# B&R Automation Studio project Lab3
Automation Studio 4.5.2.102

## Configuration SampleText

### IoMap.iom - 4PP065_0571_P74/IoMap.iom
```iecst
VAR_CONFIG
	::SDCAxisCtr:pwm_period AT %QW."X20MM4456".PeriodDurationPWM;
	::SDCAxisCtr:axis_X.pwm_value AT %QW."X20MM4456".PulseWidthCurrentPWM01;
	::SDCAxisCtr:axis_X.reset_error AT %QX."X20MM4456".ClearError01;
	::SDCAxisCtr:axis_X.reset_counter AT %QX."X20MM4456".ResetCounter01;
	::SDCAxisCtr:axis_X.counter AT %IW."X20MM4456".Counter01;
	::SDCAxisCtr:axis_X.endswitch_b_reached AT %IX."X20MM4456".StatusInput03;
	::SDCAxisCtr:axis_X.endswitch_a_reached AT %IX."X20MM4456".StatusInput04;
	::SDCAxisCtr:coil_pwm_value AT %QW."X20MM4456".PulseWidthCurrentPWM04;
	::SDCAxisCtr:axis_X.direction AT %IX."X20DI9371".DigitalInput01;
	::SDCAxisCtr:axis_X.button_b AT %IX."X20DI9371".DigitalInput02;
	::SDCAxisCtr:axis_X.button_a AT %IX."X20DI9371".DigitalInput03;
	::SDCAxisCtr:coil_powered AT %IX."X20DI9371".DigitalInput04;
	::SDCAxisCt1:axis_Y.pwm_value AT %QW."X20MM4456".PulseWidthCurrentPWM02;
	::SDCAxisCt1:axis_Y.reset_error AT %QX."X20MM4456".ClearError02;
	::SDCAxisCt1:axis_Y.reset_counter AT %QX."X20MM4456".ResetCounter02;
	::SDCAxisCt1:axis_Y.counter AT %IW."X20MM4456".Counter02;
	::SDCAxisCt1:axis_Y.endswitch_a_reached AT %IX."X20MM4456".StatusInput07;
	::SDCAxisCt1:axis_Y.endswitch_b_reached AT %IX."X20MM4456".StatusInput08;
	::SDCAxisCt2:axis_Z.pwm_value AT %QW."X20MM4456".PulseWidthCurrentPWM03;
	::SDCAxisCt2:axis_Z.reset_error AT %QX."X20MM4456".ClearError03;
	::SDCAxisCt2:axis_Z.reset_counter AT %QX."X20MM4456".ResetCounter03;
	::SDCAxisCt2:axis_Z.counter AT %IW."X20MM4456".Counter03;
	::SDCAxisCt2:axis_Z.endswitch_a_reached AT %IX."X20MM4456".StatusInput12;
	::SDCAxisCt2:axis_Z.endswitch_b_reached AT %IX."X20MM4456".StatusInput11;
END_VAR
```

### Acp10map1.ncm - 4PP065_0571_P74/Motion/Acp10map1.ncm
```
NcMapping (NcSwId=ACP10, DisabledNodesAreHidden=False)
  NcObject gAxis_X (ModuleAddress=SDC_IF1.ST1, InterfaceType=SDC, Type=ncAXIS, Channel=1, AcoposSimulation=Off, InitParameter=gAxis_X_01, AcoposParameter=gAxis_X_1, AdditionalData=CNC_Enabled="1", Disabled=FALSE, ModuleDisabled=FALSE)
  NcObject gAxis_Y (ModuleAddress=SDC_IF1.ST2, InterfaceType=SDC, Type=ncAXIS, Channel=1, AcoposSimulation=Off, InitParameter=gAxis_YZ_0, AcoposParameter=gAxis_YZ01, AdditionalData=CNC_Enabled="1", Disabled=FALSE)
  NcObject gAxis_Z (ModuleAddress=SDC_IF1.ST3, InterfaceType=SDC, Type=ncAXIS, Channel=1, AcoposSimulation=Off, InitParameter=gAxis_YZ_0, AcoposParameter=gAxis_YZ01, AdditionalData=CNC_Enabled="1", Disabled=FALSE)
```

### Arnc0map.ncm - 4PP065_0571_P74/Motion/Arnc0map.ncm
```
NcMapping (NcSwId=ARNC0)
```

### Arnc0map1.ncm - 4PP065_0571_P74/Motion/Arnc0map1.ncm
```
NcMapping (NcSwId=ARNC0, DisabledNodesAreHidden=False)
  NcObject CNCsys (Type=ncCNCSYS, Channel=1, AcoposSimulation=Off, InitParameter=CncInit, Disabled=FALSE, ModuleDisabled=FALSE)
```

## Logical view

Binary libraries used (declarations not repeated): Runtime, Operator, AsIecCon, astime, sys_lib, asstring, brsystem, AsBrStr, AsIOTime, DataObj, AsArLog, FileIO, AsArProf, AsMem, Arnc0man, Acp10man, Acp10par, NcGlobal, Acp10sim, Acp10sdc, Acp10_MC

### Global.var - Global variables
```iecst
VAR
	gAxis_X : ACP10AXIS_typ := (0);
	gAxis_X_HW : SdcHwCfg_typ := (0);
	gAxis_X_DrvIf : SdcDrvIf16_typ := (0);
	gAxis_X_DiDoIf : SdcDiDoIf_typ := (0);
	gAxis_X_EncIf : SdcEncIf16_typ := (0);
	gAxis_Y : ACP10AXIS_typ := (0);
	gAxis_Y_HW : SdcHwCfg_typ := (0);
	gAxis_Y_DrvIf : SdcDrvIf16_typ := (0);
	gAxis_Y_DiDoIf : SdcDiDoIf_typ := (0);
	gAxis_Y_EncIf : SdcEncIf16_typ := (0);
	gAxis_Z : ACP10AXIS_typ := (0);
	gAxis_Z_HW : SdcHwCfg_typ := (0);
	gAxis_Z_DrvIf : SdcDrvIf16_typ := (0);
	gAxis_Z_DiDoIf : SdcDiDoIf_typ := (0);
	gAxis_Z_EncIf : SdcEncIf16_typ := (0);
	CNCsys : ARNC0CNC_typ := (0);
END_VAR
```

### Package Logical/Libraries - Global libraries

### Library Logical/Libraries/MotrContr (ANSIC)

#### FB_Axis.c
```c
#include <bur/plctypes.h>
#ifdef __cplusplus
	extern "C"
	{
#endif
	#include "MotrContr.h"
#ifdef __cplusplus
	};
#endif
/* TODO: Add your comment here */
void FB_Axis(struct FB_Axis* inst)
{

	/*
	switch(inst->state)
	{
		case unknown:
			if (inst->endswitch_a_reached || inst->button_a)
				inst->state = A;

			if (inst->endswitch_b_reached || inst->button_b)
				inst->state = B;

			if (inst->direction)								//
				inst->state = A_dir;

			if (!inst->direction)								//
				inst->state = B_dir;

			break;

		case B:
			inst->pwm_value = 0;
			inst->reset_error = 1;

			if (!inst->button_b && !inst->endswitch_b_reached)
				inst->state = B_dir;

			if (inst->direction)								//
				inst->state = A_dir;
			break;

		case A:
			inst->pwm_value = 0;
			inst->reset_error = 1;

			if (!inst->button_a && !inst->endswitch_a_reached)
				inst->state = A_dir;

			if (!inst->direction)								//
				inst->state = B_dir;
			break;

		case A_dir:
			inst->pwm_value = inst->u / 24.0 * 32767;			//шим соответственно напряжению с регулятора
			inst->reset_error = 0;
			inst->speed = inst->u / 24.0 * 6500.0;

			if (inst->endswitch_a_reached || inst->button_a)
				inst->state = A;

			if (!inst->direction)								//
				inst->state = B_dir;

			break;

		case B_dir:
			inst->pwm_value = -inst->u / 24.0 * 32767;			//шим соответственно напряжению с регулятора
			inst->reset_error = 0;
			inst->speed = -inst->u / 24.0 * 6500.0;

			if (inst->endswitch_b_reached || inst->button_b)
				inst->state = B;

			if (inst->direction)								//
				inst->state = A_dir;

			break;
	}
	*/

	/*if (inst->endswitch_a_reached || inst->endswitch_b_reached)
	{
		inst->reset_error=1;
	}
	else
	{*/
		inst->pwm_value= inst->u / 24.0 * 32767;//шим соответственно напряжению с регулятора
		//inst->reset_error=0;
	///}
	inst->speed = inst->u / 24.0 * 6500.0;
}
```

### Data object Logical/gAxis_X/gAxis_X_01i (Ax)

#### AxInitAcp10.ax - ACP10 init object for axis
```
InitParameter (Version=5.2.1, NcSwId=ACP10)
  ACP10AXIS_typ:
    dig_in:
      level:
        reference = ncACTIV_HI
        pos_hw_end = ncACTIV_HI
        neg_hw_end = ncACTIV_HI
        trigger1 = ncACTIV_HI
        trigger2 = ncACTIV_HI
    encoder_if:
      parameter:
        count_dir = ncSTANDARD
        scaling:
          load:
            units = 1000
            rev_motor = 1
    limit:
      parameter:
        v_pos = 10000.0
        v_neg = 10000.0
        a1_pos = 10000.0
        a2_pos = 10000.0
        a1_neg = 10000.0
        a2_neg = 10000.0
        t_jolt = 0.0
        t_in_pos = 0.0
        pos_sw_end = 8388607
        neg_sw_end = -8388608
        ds_warning = 500.0
        ds_stop = 50000.0
        a_stop = 1.0E+30
        dv_stop = 0.0
        dv_stop_mode = ncOFF
    controller:
      mode = ncPOSITION
      position:
        kv = 10.0
        tn = 0.0
        t_predict = 0.0004
        t_total = 0.0004
        p_max = 10000.0
        i_max = 0.0
      speed:
        kv = 2.0
        tn = 0.0
        t_filter = 0.0
        isq_filter1:
          type = ncOFF
          a0 = 0.0
          a1 = 0.0
          b0 = 0.0
          b1 = 0.0
          b2 = 0.0
          c0_par_id = 0
          c1_par_id = 0
        isq_filter2:
          type = ncOFF
          a0 = 0.0
          a1 = 0.0
          b0 = 0.0
          b1 = 0.0
          b2 = 0.0
          c0_par_id = 0
          c1_par_id = 0
        isq_filter3:
          type = ncOFF
          a0 = 0.0
          a1 = 0.0
          b0 = 0.0
          b1 = 0.0
          b2 = 0.0
          c0_par_id = 0
          c1_par_id = 0
      uf:
        type = ncLINEAR
        auto_config = ncMOTOR_PAR
        u0 = 0.0
        un = 0.0
        fn = 50.0
        k_f_slip = 0.0
      ff:
        torque_load = 0.0
        torque_pos = 0.0
        torque_neg = 0.0
        kv_torque = 0.0
        inertia = 0.0
        t_filter_a = 0.0
    move:
      stop:
        parameter[0]:
          decel_ramp = ncA_LIMIT
          controller = ncON
        parameter[1]:
          decel_ramp = ncA_LIMIT
          controller = ncON
        parameter[2]:
          decel_ramp = ncA_LIMIT
          controller = ncON
        parameter[3]:
          decel_ramp = ncA_LIMIT
          controller = ncON
        quickstop:
          decel_ramp = ncA_LIMIT
          t_jolt = 0.0
        drive_error:
          decel_ramp = ncA_LIMIT
      homing:
        parameter:
          s = 0
          v_switch = 6000.0
          v_trigger = 2000.0
          a = 10000.0
          mode = ncEND_SWITCH
          edge_sw = ncNEGATIVE
          start_dir = ncPOSITIVE
          trigg_dir = ncNEGATIVE
          ref_pulse = ncOFF
          fix_dir = ncOFF
          tr_s_block = 0.0
          torque_lim = 0.0
          ds_block = 0.0
          ds_stop = 0.0
      basis:
        parameter:
          v_pos = 5000.0
          v_neg = 5000.0
          a1_pos = 10000.0
          a2_pos = 10000.0
          a1_neg = 10000.0
          a2_neg = 10000.0
    message:
      text:
        parameter:
          format = ncBREAK
          columns = 80
          data_modul
```

### Package Logical/gAxis_YZ - gAxis01obj

### Data object Logical/gAxis_YZ/gAxis_YZ_01a (Apt)

#### gAxis01a.apt
```
AcoposParameterTable:
  Root Parameters:
    64201 = 6500 (Name=SERVO_V_MAX_OUTPUT)
    109 = 24 (Name=SCALE_ENCOD_INCR)  // Encoder1: Encoder scaling: increments per encoder revolution
```

### Data object Logical/gAxis_YZ/gAxis_YZ_01i (Ax)

#### gAxis01i.ax
```
InitParameter (Version=5.2.1, NcSwId=ACP10)
  ACP10AXIS_typ:
    dig_in:
      level:
        reference = ncACTIV_HI
        pos_hw_end = ncACTIV_HI
        neg_hw_end = ncACTIV_HI
        trigger1 = ncACTIV_HI
        trigger2 = ncACTIV_HI
    encoder_if:
      parameter:
        count_dir = ncSTANDARD
        scaling:
          load:
            units = 3000
            rev_motor = 1
    limit:
      parameter:
        v_pos = 10000.0
        v_neg = 10000.0
        a1_pos = 10000.0
        a2_pos = 10000.0
        a1_neg = 10000.0
        a2_neg = 10000.0
        t_jolt = 0.0
        t_in_pos = 0.0
        pos_sw_end = 8388607
        neg_sw_end = -8388608
        ds_warning = 500.0
        ds_stop = 50000.0
        a_stop = 1.0E+30
        dv_stop = 0.0
        dv_stop_mode = ncOFF
    controller:
      mode = ncPOSITION
      position:
        kv = 10.0
        tn = 0.0
        t_predict = 0.0004
        t_total = 0.0004
        p_max = 1.0E+30
        i_max = 0.0
      speed:
        kv = 2.0
        tn = 0.0
        t_filter = 0.0
        isq_filter1:
          type = ncOFF
          a0 = 0.0
          a1 = 0.0
          b0 = 0.0
          b1 = 0.0
          b2 = 0.0
          c0_par_id = 0
          c1_par_id = 0
        isq_filter2:
          type = ncOFF
          a0 = 0.0
          a1 = 0.0
          b0 = 0.0
          b1 = 0.0
          b2 = 0.0
          c0_par_id = 0
          c1_par_id = 0
        isq_filter3:
          type = ncOFF
          a0 = 0.0
          a1 = 0.0
          b0 = 0.0
          b1 = 0.0
          b2 = 0.0
          c0_par_id = 0
          c1_par_id = 0
      uf:
        type = ncLINEAR
        auto_config = ncMOTOR_PAR
        u0 = 0.0
        un = 0.0
        fn = 50.0
        k_f_slip = 0.0
      ff:
        torque_load = 0.0
        torque_pos = 0.0
        torque_neg = 0.0
        kv_torque = 0.0
        inertia = 0.0
        t_filter_a = 0.0
    move:
      stop:
        parameter[0]:
          decel_ramp = ncA_LIMIT
          controller = ncON
        parameter[1]:
          decel_ramp = ncA_LIMIT
          controller = ncON
        parameter[2]:
          decel_ramp = ncA_LIMIT
          controller = ncON
        parameter[3]:
          decel_ramp = ncA_LIMIT
          controller = ncON
        quickstop:
          decel_ramp = ncA_LIMIT
          t_jolt = 0.0
        drive_error:
          decel_ramp = ncA_LIMIT
      homing:
        parameter:
          s = 0
          v_switch = 6000.0
          v_trigger = 2000.0
          a = 10000.0
          mode = ncEND_SWITCH
          edge_sw = ncNEGATIVE
          start_dir = ncPOSITIVE
          trigg_dir = ncNEGATIVE
          ref_pulse = ncOFF
          fix_dir = ncOFF
          tr_s_block = 0.0
          torque_lim = 0.0
          ds_block = 0.0
          ds_stop = 0.0
      basis:
        parameter:
          v_pos = 5000.0
          v_neg = 5000.0
          a1_pos = 10000.0
          a2_pos = 10000.0
          a1_neg = 10000.0
          a2_neg = 10000.0
    message:
      text:
        parameter:
          format = ncBREAK
          columns = 80
          data_modul
```

### Program Logical/SDCAxisCtrlX (ANSIC)

#### Cyclic.c
```c
#include <bur/plctypes.h>

#ifdef _DEFAULT_INCLUDES
	#include <AsDefault.h>
#endif

void _CYCLIC ProgramCyclic(void)
{
	gAxis_X_EncIf.iLifeCnt++;
	gAxis_X_DiDoIf.iLifeCntDriveEnable++;
	gAxis_X_DiDoIf.iLifeCntDriveReady++;
	gAxis_X_DiDoIf.iLifeCntNegHwEnd++;
	gAxis_X_DiDoIf.iLifeCntPosHwEnd++;
	gAxis_X_DiDoIf.iLifeCntReference++;
	gAxis_X_DrvIf.iLifeCnt++;

	gAxis_X_EncIf.iActTime = (INT)AsIOTimeCyclicStart();
	gAxis_X_EncIf.iActPos = - axis_X.counter;

	gAxis_X_DiDoIf.iPosHwEnd = axis_X.endswitch_a_reached;
	gAxis_X_DiDoIf.iNegHwEnd = axis_X.endswitch_b_reached;

	//coil_pwm_value = coil_powered?32767:0;
	if(coil_powered)
		coil_pwm_value = 32767;
	else
		coil_pwm_value = 0;

	//fb_controller.e = 100 * 6500.0 / 32767 - axis_X.speed; //6500.0 максимльня скорость в метках в секунду
	fb_controller.e = gAxis_X_DrvIf.oSetPos * 6500 / 32767 - axis_X.speed; //6500.0 максимльня скорость в метках в секунду
	FB_Regulator(&fb_controller); // передать значение в регулятор
	axis_X.u = fb_controller.u;

	//axis_X.u = 18;

	FB_Axis(&axis_X);
}
```

#### Init.c
```c
#include <bur/plctypes.h>

#ifdef _DEFAULT_INCLUDES
	#include <AsDefault.h>
#endif

void _INIT ProgramInit(void)
{
	//Устанавливаем типы SDC модулей
	gAxis_X_HW.EncIf1_Typ = ncSDC_ENC16;
	gAxis_X_HW.DiDoIf_Typ = ncSDC_DIDO;
	gAxis_X_HW.DrvIf_Typ = ncSDC_DRVSERVO16;
	//Устанавливаем имена переменных
	strcpy(gAxis_X_HW.EncIf1_Name, "gAxis_X_EncIf");
	strcpy(gAxis_X_HW.DrvIf_Name, "gAxis_X_DrvIf");
	strcpy(gAxis_X_HW.DiDoIf_Name, "gAxis_X_DiDoIf");
	//Устанавливаем входы готовности и нормальной работы
	gAxis_X_EncIf.iEncOK = 1;
	gAxis_X_DrvIf.iDrvOK = 1;
	gAxis_X_DrvIf.iStatusEnable = 1;
	gAxis_X_DiDoIf.iDriveReady = 1;

	fb_controller.k_p=0.0001;
	fb_controller.k_i=30;

	fb_controller.dt=0.002;
	fb_controller.integrator.dt=0.002;

	fb_controller.max_abs_value=24;

	pwm_period = 200;

	enable=1;
}
```

### Program Logical/SDCAxisCtrlY (ANSIC)

#### Variables.var
```iecst
VAR
	axis_Y : FB_Axis := (0);
	coil_powered : BOOL := FALSE;
	coil_pwm_value : INT := 0;
	fb_controller : FB_Regulator := (0);
	pwm_period : UINT := 0;
	enable : BOOL := FALSE;
END_VAR
```

#### Cyclic.c
```c
#include <bur/plctypes.h>

#ifdef _DEFAULT_INCLUDES
	#include <AsDefault.h>
#endif

void _CYCLIC ProgramCyclic(void)
{
	gAxis_Y_EncIf.iLifeCnt++;
	gAxis_Y_DiDoIf.iLifeCntDriveEnable++;
	gAxis_Y_DiDoIf.iLifeCntDriveReady++;
	gAxis_Y_DiDoIf.iLifeCntNegHwEnd++;
	gAxis_Y_DiDoIf.iLifeCntPosHwEnd++;
	gAxis_Y_DiDoIf.iLifeCntReference++;
	gAxis_Y_DrvIf.iLifeCnt++;

	gAxis_Y_EncIf.iActTime = (INT)AsIOTimeCyclicStart();
	gAxis_Y_EncIf.iActPos = axis_Y.counter;

	gAxis_Y_DiDoIf.iPosHwEnd = axis_Y.endswitch_a_reached;
	gAxis_Y_DiDoIf.iNegHwEnd = axis_Y.endswitch_b_reached;

	//coil_pwm_value = coil_powered?32767:0;
	if(coil_powered)
		coil_pwm_value = 32767;
	else
		coil_pwm_value = 0;

	//fb_controller.e = 100 * 6500.0 / 32767 - axis_X.speed; //6500.0 максимльня скорость в метках в секунду
	fb_controller.e = gAxis_Y_DrvIf.oSetPos * 6500 / 32767 - axis_Y.speed; //6500.0 максимльня скорость в метках в секунду
	FB_Regulator(&fb_controller); // передать значение в регулятор
	axis_Y.u = fb_controller.u;

	//axis_X.u = 18;

	FB_Axis(&axis_Y);
}
```

#### Init.c
```c
#include <bur/plctypes.h>

#ifdef _DEFAULT_INCLUDES
	#include <AsDefault.h>
#endif

void _INIT ProgramInit(void)
{
	//Устанавливаем типы SDC модулей
	gAxis_Y_HW.EncIf1_Typ = ncSDC_ENC16;
	gAxis_Y_HW.DiDoIf_Typ = ncSDC_DIDO;
	gAxis_Y_HW.DrvIf_Typ = ncSDC_DRVSERVO16;
	//Устанавливаем имена переменных
	strcpy(gAxis_Y_HW.EncIf1_Name, "gAxis_Y_EncIf");
	strcpy(gAxis_Y_HW.DrvIf_Name, "gAxis_Y_DrvIf");
	strcpy(gAxis_Y_HW.DiDoIf_Name, "gAxis_Y_DiDoIf");
	//Устанавливаем входы готовности и нормальной работы
	gAxis_Y_EncIf.iEncOK = 1;
	gAxis_Y_DrvIf.iDrvOK = 1;
	gAxis_Y_DrvIf.iStatusEnable = 1;
	gAxis_Y_DiDoIf.iDriveReady = 1;

	fb_controller.k_p=0.002;
	fb_controller.k_i=0.16;

	fb_controller.dt=0.002;
	fb_controller.integrator.dt=0.002;

	fb_controller.max_abs_value=24;

	pwm_period = 200;

	enable=1;
}
```

### Program Logical/SDCAxisCtrlZ (ANSIC)

#### Variables.var
```iecst
VAR
	axis_Z : FB_Axis := (0);
	coil_powered : BOOL := FALSE;
	coil_pwm_value : INT := 0;
	fb_controller : FB_Regulator := (0);
	pwm_period : UINT := 0;
	enable : BOOL := FALSE;
END_VAR
```

#### Cyclic.c
```c
#include <bur/plctypes.h>

#ifdef _DEFAULT_INCLUDES
	#include <AsDefault.h>
#endif

void _CYCLIC ProgramCyclic(void)
{
	gAxis_Z_EncIf.iLifeCnt++;
	gAxis_Z_DiDoIf.iLifeCntDriveEnable++;
	gAxis_Z_DiDoIf.iLifeCntDriveReady++;
	gAxis_Z_DiDoIf.iLifeCntNegHwEnd++;
	gAxis_Z_DiDoIf.iLifeCntPosHwEnd++;
	gAxis_Z_DiDoIf.iLifeCntReference++;
	gAxis_Z_DrvIf.iLifeCnt++;

	gAxis_Z_EncIf.iActTime = (INT)AsIOTimeCyclicStart();
	gAxis_Z_EncIf.iActPos = axis_Z.counter;

	gAxis_Z_DiDoIf.iPosHwEnd = axis_Z.endswitch_a_reached;
	gAxis_Z_DiDoIf.iNegHwEnd = axis_Z.endswitch_b_reached;

	//coil_pwm_value = coil_powered?32767:0;
	if(coil_powered)
		coil_pwm_value = 32767;
	else
		coil_pwm_value = 0;

	//fb_controller.e = 100 * 6500.0 / 32767 - axis_X.speed; //6500.0 максимльня скорость в метках в секунду
	fb_controller.e = gAxis_Z_DrvIf.oSetPos * 6500 / 32767 - axis_Z.speed; //6500.0 максимльня скорость в метках в секунду
	FB_Regulator(&fb_controller); // передать значение в регулятор
	axis_Z.u = fb_controller.u;

	//axis_X.u = 18;

	FB_Axis(&axis_Z);
}
```

#### Init.c
```c
#include <bur/plctypes.h>

#ifdef _DEFAULT_INCLUDES
	#include <AsDefault.h>
#endif

void _INIT ProgramInit(void)
{
	//Устанавливаем типы SDC модулей
	gAxis_Z_HW.EncIf1_Typ = ncSDC_ENC16;
	gAxis_Z_HW.DiDoIf_Typ = ncSDC_DIDO;
	gAxis_Z_HW.DrvIf_Typ = ncSDC_DRVSERVO16;
	//Устанавливаем имена переменных
	strcpy(gAxis_Z_HW.EncIf1_Name, "gAxis_Z_EncIf");
	strcpy(gAxis_Z_HW.DrvIf_Name, "gAxis_Z_DrvIf");
	strcpy(gAxis_Z_HW.DiDoIf_Name, "gAxis_Z_DiDoIf");
	//Устанавливаем входы готовности и нормальной работы
	gAxis_Z_EncIf.iEncOK = 1;
	gAxis_Z_DrvIf.iDrvOK = 1;
	gAxis_Z_DrvIf.iStatusEnable = 1;
	gAxis_Z_DiDoIf.iDriveReady = 1;

	fb_controller.k_p=0.002;
	fb_controller.k_i=0.16;

	fb_controller.dt=0.002;
	fb_controller.integrator.dt=0.002;

	fb_controller.max_abs_value=24;

	pwm_period = 200;

	enable=1;
}
```

### Data object Logical/CncInit (Cns)

- CncInit.cns (not shown)

### Data object Logical/CncProg (Cnc)

#### CncProg.cnc
```
%001 (CncProgram)

( TODO: Add code here )

N10 F300000
N20 G01 X0 Y100000
N30 G01 X0 Y100000 Z100000
N40 G01 X66700 Y0 Z100000
N50 G01 X0 Y0 Z100000
N60 G01 X0 Y0 Z0

N999 M30
```

### Data object Logical/test (Cnc)

#### CncProg.cnc
```
%001 (CncProgram)

( TODO: Add code here )

N10 F300000
N20 G01 X66700 Y100000 Z100000

N999 M30
```

### Data object Logical/test1 (Cnc)

#### CncProg.cnc
```
%001 (CncProgram)

( TODO: Add code here )

N10 F300000
N20 G01 X0 Y0 Z0

N999 M30
```

Listed in the project but not available here: Logical/Global.typ, Logical/acp10etxen, Logical/gAxis_X/gAxis_X_01a, Logical/GmcIpConfig, Logical/GmcIpUserConfig
